ORGANIZATION_BLOCK "Connect"
TITLE = "Main Program Sweep (Cycle)"
{ S7_Optimized_Access := 'TRUE' }
VERSION : 0.1

BEGIN
END_ORGANIZATION_BLOCK

